FUNCTION_BLOCK Tank_Fault EXTENDS _Tank_State

METHOD OnExecute
IF _ctx.hmi.bResetButton THEN
	_ctx.hmi.bResetButton := FALSE;
	_ctx.priv.smgr.Request(_ctx.state.iDisabled);
END_IF
END_METHOD

METHOD OnInit
_ctx.io.out.bInletValveOpen := FALSE;
_ctx.hmi.bResetButtonVis := TRUE;
_ctx.priv.IsFillable.Lower();
END_METHOD

END_FUNCTION_BLOCK

(* stored: Version 1.1.0.1
   POU Tank_Fault: Id {745d540a-e4c5-469b-a1d3-4ffa631c010d}, SpecialFunc None
   Method OnExecute: Id {06b2ad95-f7be-4415-9c3c-55c1d733a073}
   Method OnInit: Id {4892cd4f-4c2d-48c7-903e-7629ffdbab56} *)
